PROGRAM P_ADS_Screw
VAR
	bTrigger				: BOOL;
		
//pliki zakręcarek
	fbRead_19:	FB_ReadAdsSymByName;
	AStChartGripperScrewer1	:ARRAY[0..100] OF ARRAY[0..5, 0..500] OF INT;
	fbCyclicReadout: TON;
	
	fbRead_20:	FB_ReadAdsSymByName;
	bScrewer1Done1 :BOOL;
	bScrewer1Done2 :BOOL;
	fbRead_21:	FB_ReadAdsSymByName;
	bScrewer2Done1 :BOOL;
	bScrewer2Done2 :BOOL;
	fbRead_22:	FB_ReadAdsSymByName;
	fbRead_23:	FB_ReadAdsSymByName;
	fbRead_24:	FB_ReadAdsSymByName;
	fbRead_25:	FB_ReadAdsSymByName;
	fbRead_26:	FB_ReadAdsSymByName;
	AStChartGripperScrewer2	:ARRAY[0..100] OF ARRAY[0..5, 0..500] OF INT;
	bScrewer1NotDone1 :BOOL;
	bScrewer2NotDone1 :BOOL;
	bScrewer1Run:BOOL;
	bScrewer2Run:BOOL;
	fbRead_27:	FB_ReadAdsSymByName;
	fbRead_28:	FB_ReadAdsSymByName;
	fbRead_29:	FB_ReadAdsSymByName;
	fbRead_30:	FB_ReadAdsSymByName;	
	lrGripperScrewer1TorqueCV :LREAL;
	lrGripperScrewer2TorqueCV :LREAL;
	fbRead_31:	FB_ReadAdsSymByName;
	fbRead_32:	FB_ReadAdsSymByName;
	lrGripperScrewingTightTorqueShow:LREAL;
	lrGripperScrewing2TightTorqueShow:LREAL;
END_VAR

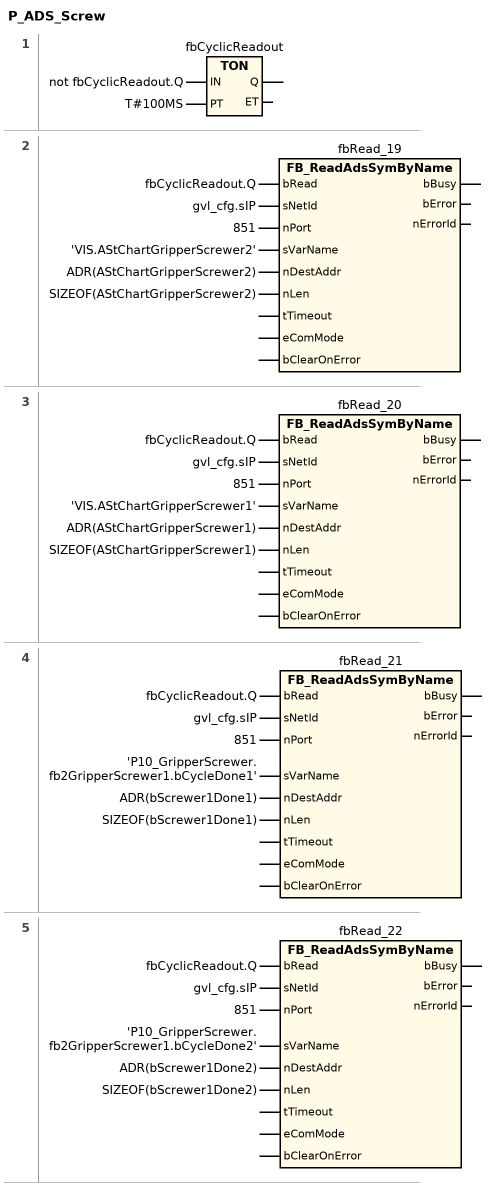
// NETWORK 1
fbCyclicReadout(IN := not fbCyclicReadout.Q, PT := T#100MS); // TON

// NETWORK 2
fbRead_19(
    bRead := fbCyclicReadout.Q,
    sNetId := gvl_cfg.sIP,
    nPort := 851,
    sVarName := 'VIS.AStChartGripperScrewer2',
    nDestAddr := ADR(AStChartGripperScrewer2),
    nLen := SIZEOF(AStChartGripperScrewer2)); // FB_ReadAdsSymByName

// NETWORK 3
fbRead_20(
    bRead := fbCyclicReadout.Q,
    sNetId := gvl_cfg.sIP,
    nPort := 851,
    sVarName := 'VIS.AStChartGripperScrewer1',
    nDestAddr := ADR(AStChartGripperScrewer1),
    nLen := SIZEOF(AStChartGripperScrewer1)); // FB_ReadAdsSymByName

// NETWORK 4
fbRead_21(
    bRead := fbCyclicReadout.Q,
    sNetId := gvl_cfg.sIP,
    nPort := 851,
    sVarName := 'P10_GripperScrewer.fb2GripperScrewer1.bCycleDone1',
    nDestAddr := ADR(bScrewer1Done1),
    nLen := SIZEOF(bScrewer1Done1)); // FB_ReadAdsSymByName

// NETWORK 5
fbRead_22(
    bRead := fbCyclicReadout.Q,
    sNetId := gvl_cfg.sIP,
    nPort := 851,
    sVarName := 'P10_GripperScrewer.fb2GripperScrewer1.bCycleDone2',
    nDestAddr := ADR(bScrewer1Done2),
    nLen := SIZEOF(bScrewer1Done2)); // FB_ReadAdsSymByName

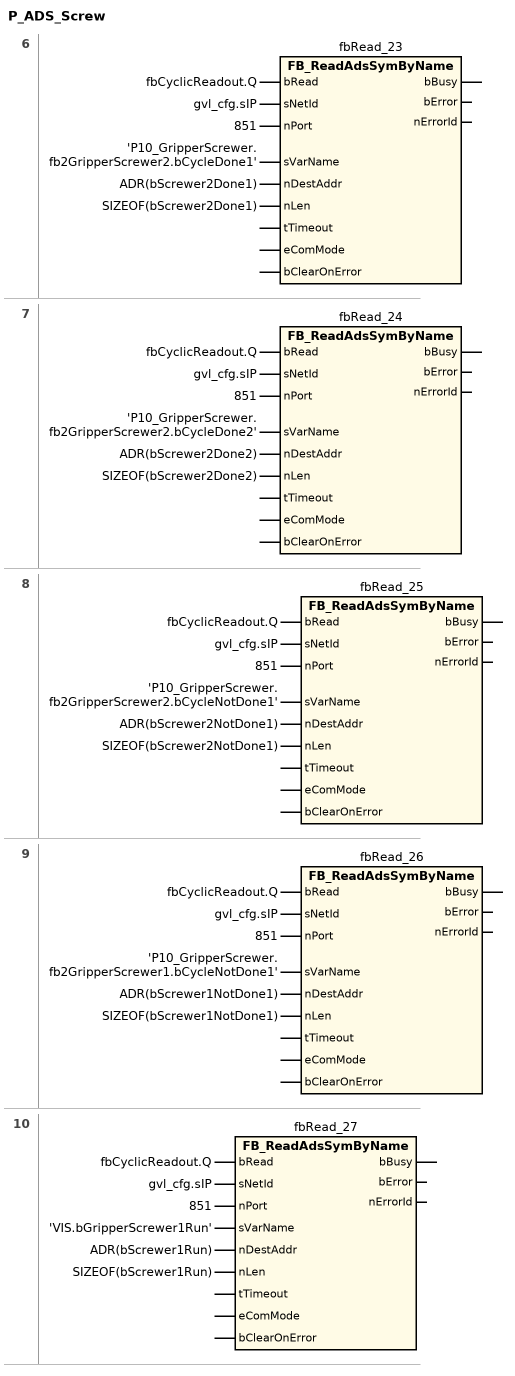
// NETWORK 6
fbRead_23(
    bRead := fbCyclicReadout.Q,
    sNetId := gvl_cfg.sIP,
    nPort := 851,
    sVarName := 'P10_GripperScrewer.fb2GripperScrewer2.bCycleDone1',
    nDestAddr := ADR(bScrewer2Done1),
    nLen := SIZEOF(bScrewer2Done1)); // FB_ReadAdsSymByName

// NETWORK 7
fbRead_24(
    bRead := fbCyclicReadout.Q,
    sNetId := gvl_cfg.sIP,
    nPort := 851,
    sVarName := 'P10_GripperScrewer.fb2GripperScrewer2.bCycleDone2',
    nDestAddr := ADR(bScrewer2Done2),
    nLen := SIZEOF(bScrewer2Done2)); // FB_ReadAdsSymByName

// NETWORK 8
fbRead_25(
    bRead := fbCyclicReadout.Q,
    sNetId := gvl_cfg.sIP,
    nPort := 851,
    sVarName := 'P10_GripperScrewer.fb2GripperScrewer2.bCycleNotDone1',
    nDestAddr := ADR(bScrewer2NotDone1),
    nLen := SIZEOF(bScrewer2NotDone1)); // FB_ReadAdsSymByName

// NETWORK 9
fbRead_26(
    bRead := fbCyclicReadout.Q,
    sNetId := gvl_cfg.sIP,
    nPort := 851,
    sVarName := 'P10_GripperScrewer.fb2GripperScrewer1.bCycleNotDone1',
    nDestAddr := ADR(bScrewer1NotDone1),
    nLen := SIZEOF(bScrewer1NotDone1)); // FB_ReadAdsSymByName

// NETWORK 10
fbRead_27(
    bRead := fbCyclicReadout.Q,
    sNetId := gvl_cfg.sIP,
    nPort := 851,
    sVarName := 'VIS.bGripperScrewer1Run',
    nDestAddr := ADR(bScrewer1Run),
    nLen := SIZEOF(bScrewer1Run)); // FB_ReadAdsSymByName

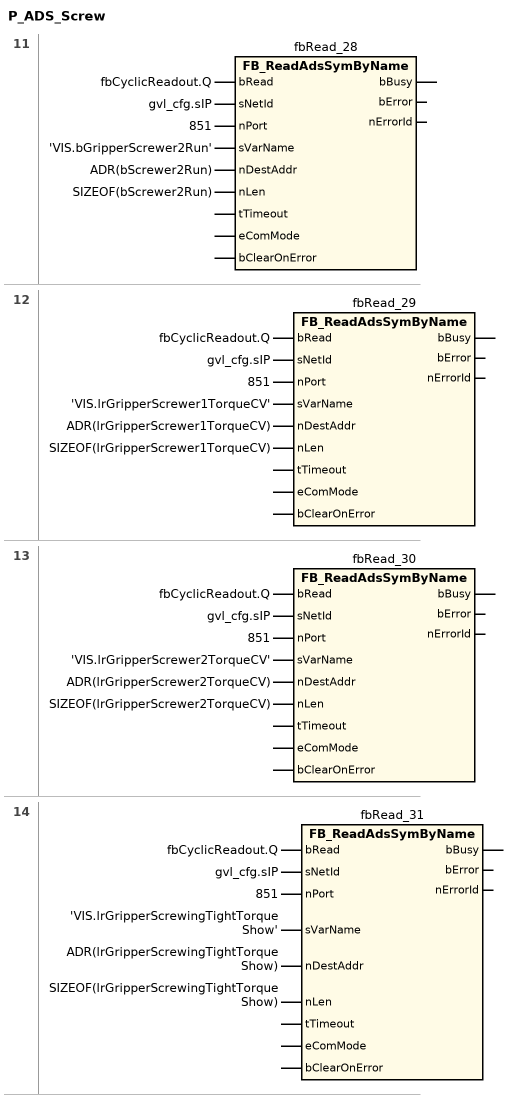
// NETWORK 11
fbRead_28(
    bRead := fbCyclicReadout.Q,
    sNetId := gvl_cfg.sIP,
    nPort := 851,
    sVarName := 'VIS.bGripperScrewer2Run',
    nDestAddr := ADR(bScrewer2Run),
    nLen := SIZEOF(bScrewer2Run)); // FB_ReadAdsSymByName

// NETWORK 12
fbRead_29(
    bRead := fbCyclicReadout.Q,
    sNetId := gvl_cfg.sIP,
    nPort := 851,
    sVarName := 'VIS.lrGripperScrewer1TorqueCV',
    nDestAddr := ADR(lrGripperScrewer1TorqueCV),
    nLen := SIZEOF(lrGripperScrewer1TorqueCV)); // FB_ReadAdsSymByName

// NETWORK 13
fbRead_30(
    bRead := fbCyclicReadout.Q,
    sNetId := gvl_cfg.sIP,
    nPort := 851,
    sVarName := 'VIS.lrGripperScrewer2TorqueCV',
    nDestAddr := ADR(lrGripperScrewer2TorqueCV),
    nLen := SIZEOF(lrGripperScrewer2TorqueCV)); // FB_ReadAdsSymByName

// NETWORK 14
fbRead_31(
    bRead := fbCyclicReadout.Q,
    sNetId := gvl_cfg.sIP,
    nPort := 851,
    sVarName := 'VIS.lrGripperScrewingTightTorqueShow',
    nDestAddr := ADR(lrGripperScrewingTightTorqueShow),
    nLen := SIZEOF(lrGripperScrewingTightTorqueShow)); // FB_ReadAdsSymByName

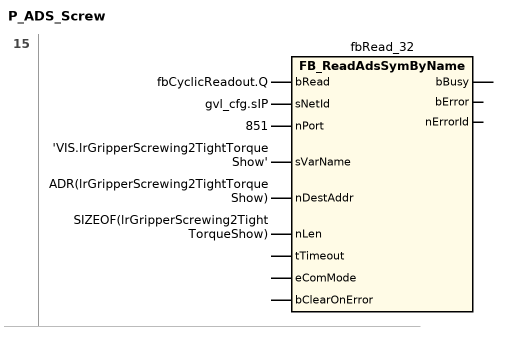
// NETWORK 15
fbRead_32(
    bRead := fbCyclicReadout.Q,
    sNetId := gvl_cfg.sIP,
    nPort := 851,
    sVarName := 'VIS.lrGripperScrewing2TightTorqueShow',
    nDestAddr := ADR(lrGripperScrewing2TightTorqueShow),
    nLen := SIZEOF(lrGripperScrewing2TightTorqueShow)); // FB_ReadAdsSymByName

END_PROGRAM

(* stored: Version 1.2.0.0, ProductVersion 3.1.4026.13, FileIdentifier 11d0cf8b27c9ec5eab59b1062a3e820cd4f3bb7b, FileSignature 94b75b0682bbe25184a02cef1e8cddaf0bf2af5b7ed1ae71fc067d391b1627eefb6ba7285e9373f37960611f74f3364ed86b82def921bfb359f15f1b668ec2b20c88972381a7e3a8a021b5efdca71008d2a0ab4c7c49a735e32a9f71d7ffa801eb8906a3b9f915df5b494b0084f8db2c5c11eb5f80885dcaa74d3c770f0adfb9871c61c5e94e276ff01d76498d4bd2106e7a25d578657c435cd675e4f1b06059de54887211b1f85fad1a0ba4025710e96ae5a5505981e576a747e23da57cd4b92c5c99d9f80da03ffd04383ae604275a08c1d8e1983c30b407bdaf4cc1b718411a31535837bfe053d435604e6750fec05f8fbf920a680527fa598f15fd350950
   POU P_ADS_Screw: Id {d7214866-d5f3-4296-b0b8-db821db6c1c7}, SpecialFunc None *)
